(* LS Electric XG5000 project: Eyasin_Clone_Shaon *)
(* PLC LSPLC *)

PROGRAM NewProgram (* task: Scan Program *)
VAR
    BOSS : BOOL;
    CONVAYOR : BOOL;
    CONV_M AT %QX0.0.6 : BOOL;
    CS1 AT %IX0.0.0 : BOOL;
    CS2 : BOOL;
    CS3 AT %IX0.0.2 : BOOL;
    CS4 : BOOL;
    CS5 AT %IX0.0.4 : BOOL;
    CS6 AT %IX0.0.5 : BOOL;
    CS7 AT %IX0.0.6 : BOOL;
    CS8 AT %IX0.0.7 : BOOL;
    DRILL_M AT %QX0.0.5 : BOOL;
    DRILL_T_IN : BOOL;
    DRILL_UP : BOOL;
    EJECTER_OK : BOOL;
    EJECTER_RET : BOOL;
    GL AT %QX0.0.9 : BOOL;
    INST : TON;
    INST1 : TON;
    METAL_T_IN : BOOL;
    RL AT %QX0.0.7 : BOOL;
    S1 : BOOL;
    S2 : BOOL;
    S3 : BOOL;
    S4 : BOOL;
    S5 : BOOL;
    SAN_2 AT %IX0.0.9 : BOOL;
    SAN_3 AT %IX0.0.10 : BOOL;
    SOL_1 AT %QX0.0.0 : BOOL;
    SOL_2 AT %QX0.0.1 : BOOL;
    SOL_3 AT %QX0.0.2 : BOOL;
    SOL_4 AT %QX0.0.3 : BOOL;
    SOL_5 AT %QX0.0.4 : BOOL;
    START_PB AT %IX0.0.12 : BOOL;
    STOP_PB AT %IX0.0.13 : BOOL;
    TIMER_1 : TON;
    TIMER_2 : TON;
    TIMER_3 : TOF;
    TRANSFER_RET : BOOL;
    WORK_PIECE_DETECT : BOOL;
END_VAR

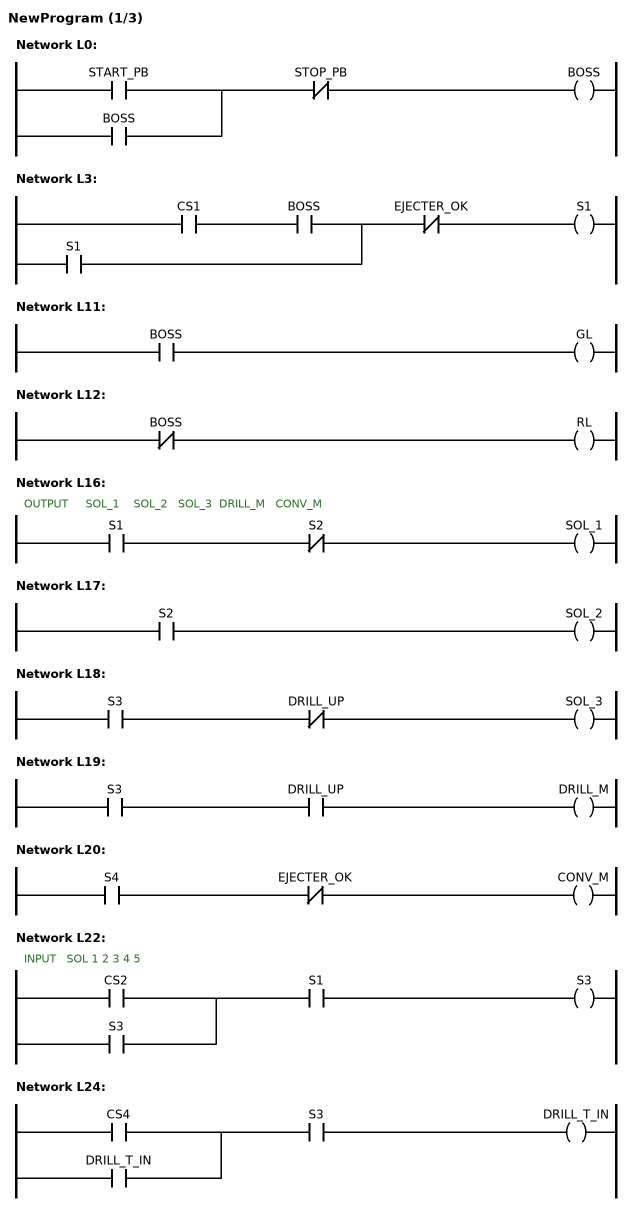
(* Rung L0 *)
BOSS := (START_PB OR BOSS) AND NOT STOP_PB;
(* Rung L3 *)
S1 := ((CS1 AND BOSS) OR S1) AND NOT EJECTER_OK;
(* Rung L11 *)
GL := BOSS;
(* Rung L12 *)
RL := NOT BOSS;
(* OUTPUT     SOL_1    SOL_2   SOL_3  DRILL_M   CONV_M *)
(* Rung L16 *)
SOL_1 := S1 AND NOT S2;
(* Rung L17 *)
SOL_2 := S2;
(* Rung L18 *)
SOL_3 := S3 AND NOT DRILL_UP;
(* Rung L19 *)
DRILL_M := S3 AND DRILL_UP;
(* Rung L20 *)
CONV_M := S4 AND NOT EJECTER_OK;
(* INPUT   SOL 1 2 3 4 5 *)
(* Rung L22 *)
S3 := (CS2 OR S3) AND S1;
(* Rung L24 *)
DRILL_T_IN := (CS4 OR DRILL_T_IN) AND S3;

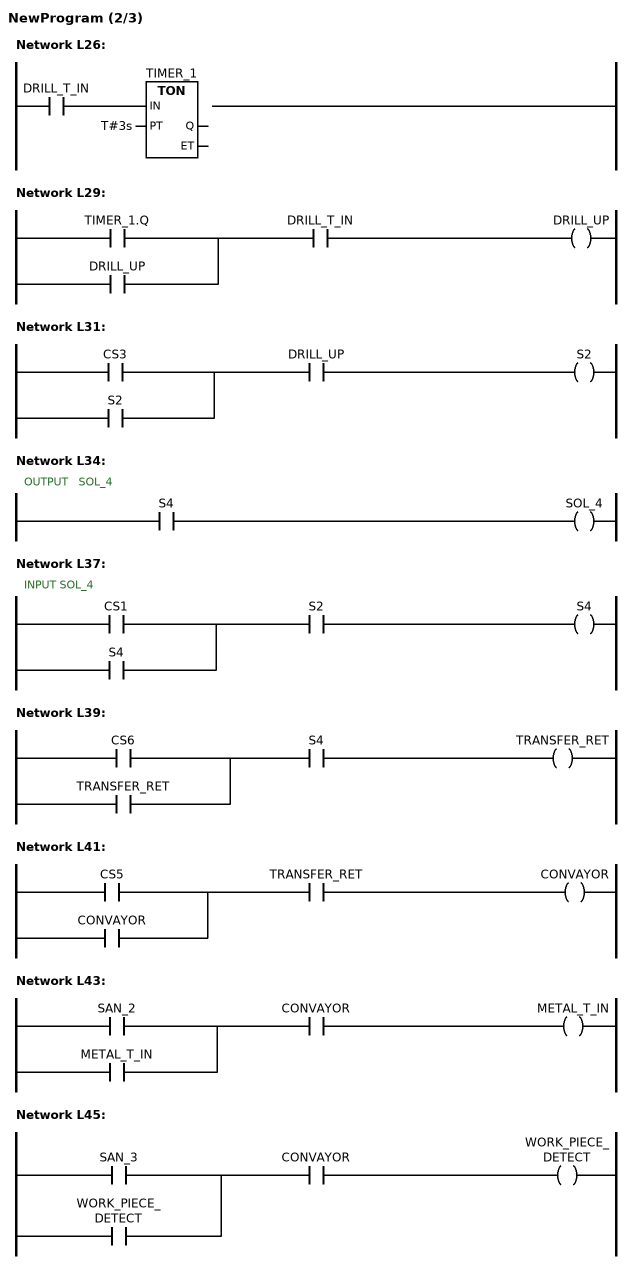
(* Rung L26 *)
TIMER_1(IN := DRILL_T_IN, PT := T#3s);
(* Rung L29 *)
DRILL_UP := (TIMER_1.Q OR DRILL_UP) AND DRILL_T_IN;
(* Rung L31 *)
S2 := (CS3 OR S2) AND DRILL_UP;
(* OUTPUT   SOL_4 *)
(* Rung L34 *)
SOL_4 := S4;
(* INPUT SOL_4 *)
(* Rung L37 *)
S4 := (CS1 OR S4) AND S2;
(* Rung L39 *)
TRANSFER_RET := (CS6 OR TRANSFER_RET) AND S4;
(* Rung L41 *)
CONVAYOR := (CS5 OR CONVAYOR) AND TRANSFER_RET;
(* Rung L43 *)
METAL_T_IN := (SAN_2 OR METAL_T_IN) AND CONVAYOR;
(* Rung L45 *)
WORK_PIECE_DETECT := (SAN_3 OR WORK_PIECE_DETECT) AND CONVAYOR;

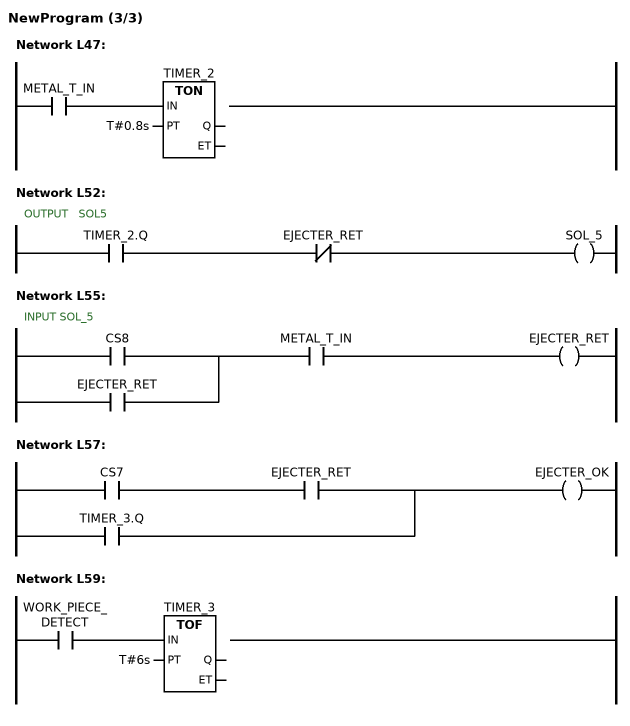
(* Rung L47 *)
TIMER_2(IN := METAL_T_IN, PT := T#0.8s);
(* OUTPUT   SOL5 *)
(* Rung L52 *)
SOL_5 := TIMER_2.Q AND NOT EJECTER_RET;
(* INPUT SOL_5 *)
(* Rung L55 *)
EJECTER_RET := (CS8 OR EJECTER_RET) AND METAL_T_IN;
(* Rung L57 *)
EJECTER_OK := (CS7 AND EJECTER_RET) OR TIMER_3.Q;
(* Rung L59 *)
TIMER_3(IN := WORK_PIECE_DETECT, PT := T#6s);
END_PROGRAM